// TIA Portal V17 export
// export: Created 2024-09-04T07:59:27.7824984Z, ExportSetting None, DisplayName Totally Integrated Automation Portal, DisplayVersion V17 Update 7, DisplayName TIA Portal Openness, DisplayVersion V17 Update 7, DisplayName TIA Portal Version Control Interface, DisplayVersion V17, DisplayName SINAMICS Startdrive Advanced, DisplayVersion V17 SP2, DisplayName SINAMICS Startdrive G110M, G120, G120C, G120D, G120P, G115D, DisplayVersion V17 SP2, DisplayName SINAMICS Startdrive G130, G150, S120, S150, SINAMICS MV, S210, DisplayVersion V17 SP2, DisplayName STEP 7 Professional, DisplayVersion V17 Update 7, DisplayName STEP 7 Safety, DisplayVersion V17 Update 6, DisplayName WinCC Professional, DisplayVersion V17 Update 7
FUNCTION_BLOCK "Block_1"   // FB12, LAD
{ S7_Optimized_Access := 'TRUE' }
// stored: MemoryReserve 100, SetENOAutomatically false
BEGIN

REGION Network 1
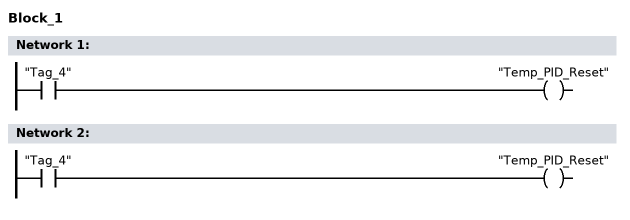
   RUNG wire#powerrail
      Contact( "Tag_4" )
      Coil( "Temp_PID_Reset" )
   END_RUNG
   // the same network as SCL:
   "Temp_PID_Reset" := "Tag_4";
END_REGION

REGION Network 2
   RUNG wire#powerrail
      Contact( "Tag_4" )
      Coil( "Temp_PID_Reset" )
   END_RUNG
   // the same network as SCL:
   "Temp_PID_Reset" := "Tag_4";
END_REGION
END_FUNCTION_BLOCK
